{attribute wpf [Container(Layout.Wrap)]}
{attribute wpf [Group(Layout.GroupBox)]}
FUNCTION_BLOCK fbDigitalSensor
VAR_INPUT
	{attribute 'hide'}
	Signal : BOOL;
END_VAR
VAR_OUTPUT
END_VAR
VAR
	{attribute wpf [Container(Layout.UniformGrid)]}
	{attribute addProperty Name "Value"}
	{attribute addProperty ToolTip "Sensor actual value"}
	Value : BOOL;
END_VAR

Value := Signal;

METHOD IsOff : BOOL
VAR_INPUT
END_VAR
Value := Signal;

IsOff := NOT Value;
END_METHOD

METHOD IsOn : BOOL
VAR_INPUT
END_VAR
Value := Signal;

IsOn := Value;
END_METHOD

END_FUNCTION_BLOCK

(* stored: Version 1.1.0.1, ProductVersion 3.1.4024.2
   POU fbDigitalSensor: Id {357a6570-1163-4d42-b43c-5cd98bab1dac}, SpecialFunc None
   Method IsOff: Id {6efed94f-c685-4163-9504-212d4b08b3cc}
   Method IsOn: Id {e42e129b-fd03-4a9e-afd9-23ccb7c8924d} *)
